// Mitsubishi GX Works2 project: e06   PLC: Q02/Q02H

PROGRAM MAIN
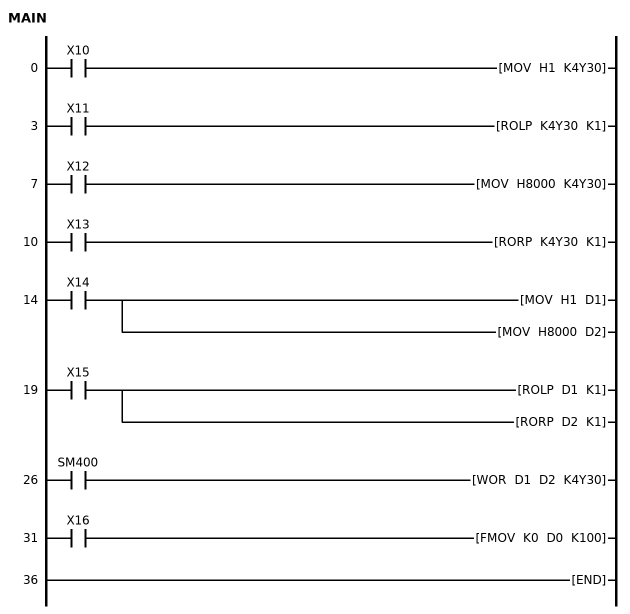
0     LD      X10
      MOV     H1 K4Y30
3     LD      X11
      ROLP    K4Y30 K1
7     LD      X12
      MOV     H8000 K4Y30
10    LD      X13
      RORP    K4Y30 K1
14    LD      X14
      MOV     H1 D1
      MOV     H8000 D2
19    LD      X15
      ROLP    D1 K1
      RORP    D2 K1
26    LD      SM400
      WOR     D1 D2 K4Y30
31    LD      X16
      FMOV    K0 D0 K100
36    END
END_PROGRAM
